FUNCTION_BLOCK LoadSensor (* Sensor for receiving data from the LoadSensor plugin controller in Polysun *)
  (* Standard: 61499-2 *)
  (* Version 1.0, 2017-07-21, Marc Jakobi, HTW Berlin *)
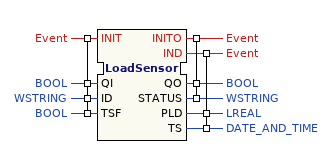
  EVENT_INPUT
    INIT WITH QI, ID, TSF; (* Initialization Request *)
  END_EVENT
  EVENT_OUTPUT
    INITO WITH QO, STATUS; (* Initialization Confirm *)
    IND WITH PLD, TS; (* Execution Confirmation *)
  END_EVENT
  VAR_INPUT
    QI : BOOL; (* Input event qualifier *)
    ID : WSTRING; (* Connection identifier *)
    TSF : BOOL; (* Flag for whether to receive time stamp or not *)
  END_VAR
  VAR_OUTPUT
    QO : BOOL; (* Output event qualifier *)
    STATUS : WSTRING; (* Service status *)
    PLD : LREAL; (* PV power output AC in W *)
    TS : DATE_AND_TIME; (* Time stamp (optional) *)
  END_VAR
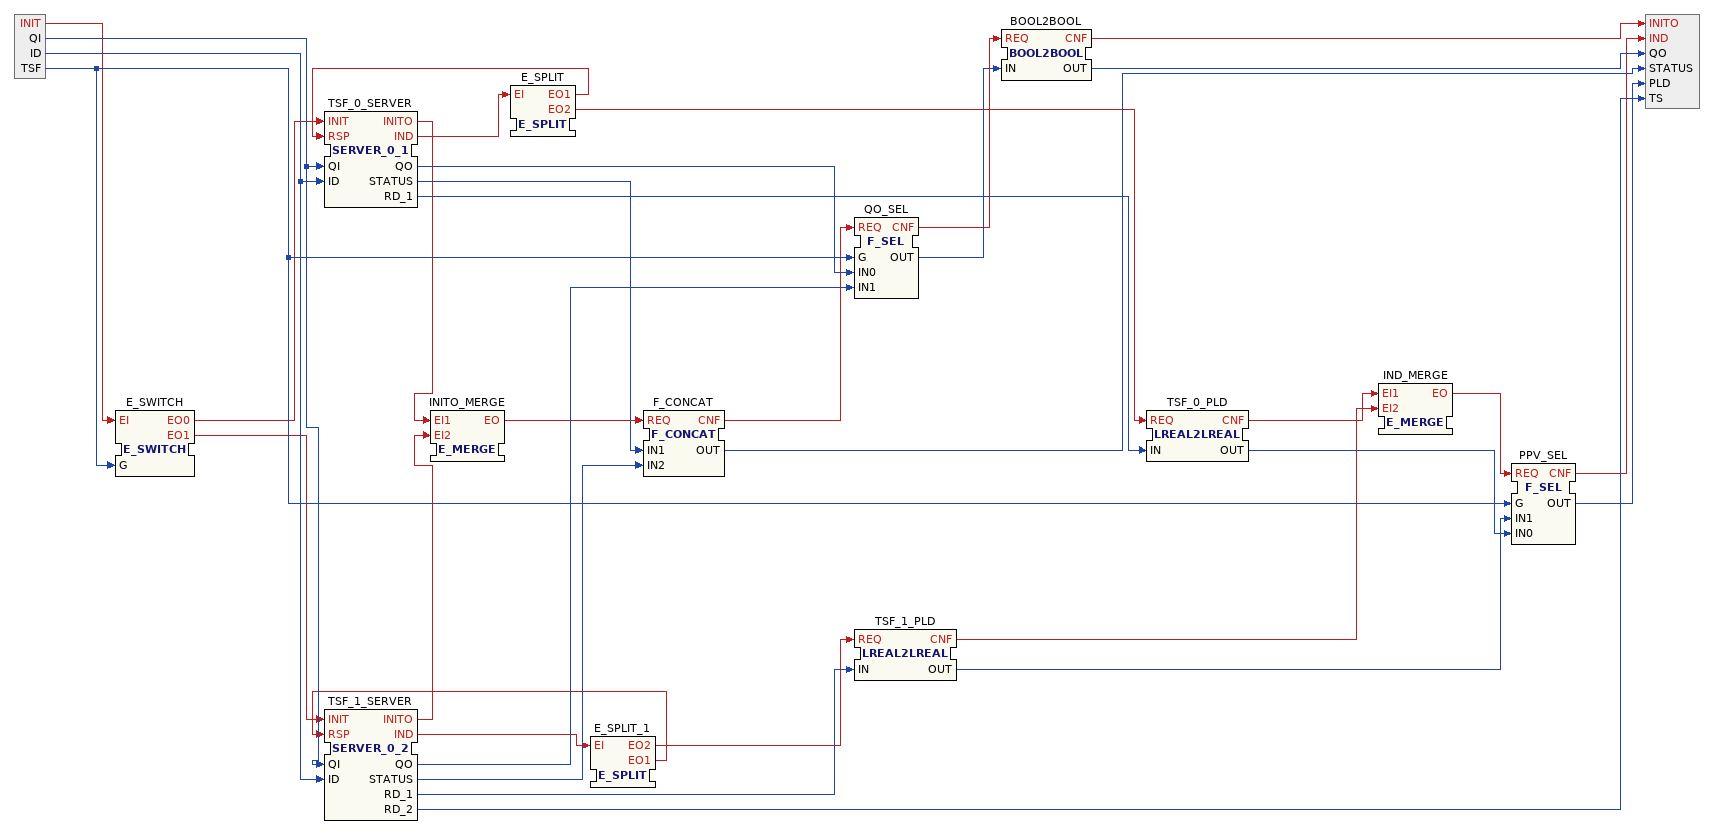
  FBS
    E_SWITCH : E_SWITCH;
    E_SPLIT : E_SPLIT;
    E_SPLIT_1 : E_SPLIT;
    INITO_MERGE : E_MERGE;
    IND_MERGE : E_MERGE;
    QO_SEL : F_SEL;
    PPV_SEL : F_SEL;
    TSF_1_PLD : LREAL2LREAL;
    TSF_0_PLD : LREAL2LREAL;
    BOOL2BOOL : BOOL2BOOL;
    F_CONCAT : F_CONCAT;
    TSF_0_SERVER : SERVER_0_1;
    TSF_1_SERVER : SERVER_0_2;
  END_FBS
  EVENT_CONNECTIONS
    INIT TO E_SWITCH.EI;
    E_SPLIT_1.EO2 TO TSF_1_PLD.REQ;
    TSF_0_PLD.CNF TO IND_MERGE.EI1;
    IND_MERGE.EO TO PPV_SEL.REQ;
    QO_SEL.CNF TO BOOL2BOOL.REQ;
    INITO_MERGE.EO TO F_CONCAT.REQ;
    F_CONCAT.CNF TO QO_SEL.REQ;
    BOOL2BOOL.CNF TO INITO;
    E_SWITCH.EO0 TO TSF_0_SERVER.INIT;
    E_SPLIT.EO1 TO TSF_0_SERVER.RSP;
    TSF_0_SERVER.INITO TO INITO_MERGE.EI1;
    TSF_0_SERVER.IND TO E_SPLIT.EI;
    E_SWITCH.EO1 TO TSF_1_SERVER.INIT;
    E_SPLIT_1.EO1 TO TSF_1_SERVER.RSP;
    TSF_1_SERVER.INITO TO INITO_MERGE.EI2;
    TSF_1_SERVER.IND TO E_SPLIT_1.EI;
    E_SPLIT.EO2 TO TSF_0_PLD.REQ;
    TSF_1_PLD.CNF TO IND_MERGE.EI2;
    PPV_SEL.CNF TO IND;
  END_CONNECTIONS
  DATA_CONNECTIONS
    TSF TO E_SWITCH.G;
    TSF TO QO_SEL.G;
    TSF TO PPV_SEL.G;
    TSF_1_PLD.OUT TO PPV_SEL.IN1;
    PPV_SEL.OUT TO PLD;
    QO_SEL.OUT TO BOOL2BOOL.IN;
    BOOL2BOOL.OUT TO QO;
    F_CONCAT.OUT TO STATUS;
    QI TO TSF_0_SERVER.QI;
    ID TO TSF_0_SERVER.ID;
    TSF_0_SERVER.QO TO QO_SEL.IN0;
    TSF_0_SERVER.STATUS TO F_CONCAT.IN1;
    QI TO TSF_1_SERVER.QI;
    ID TO TSF_1_SERVER.ID;
    TSF_1_SERVER.QO TO QO_SEL.IN1;
    TSF_1_SERVER.STATUS TO F_CONCAT.IN2;
    TSF_1_SERVER.RD_1 TO TSF_1_PLD.IN;
    TSF_1_SERVER.RD_2 TO TS;
    TSF_0_SERVER.RD_1 TO TSF_0_PLD.IN;
    TSF_0_PLD.OUT TO PPV_SEL.IN0;
  END_CONNECTIONS
END_FUNCTION_BLOCK
